FUNCTION_BLOCK ProductionRateFbt (* Composite Function Block Type *)
  (* Standard: 61499-2 *)
  (* Version 0.0, 2018-10-14, 4DIAC-IDE, 4DIAC-Consortium *)
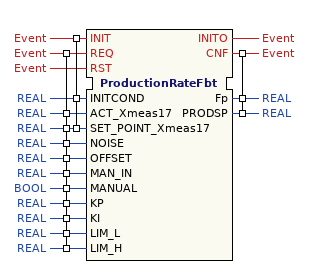
  EVENT_INPUT
    INIT WITH INITCOND, SET_POINT_Xmeas17; (* Initialization Request *)
    REQ WITH ACT_Xmeas17, SET_POINT_Xmeas17, NOISE, OFFSET, MAN_IN, MANUAL, KP, KI, LIM_L, LIM_H; (* Normal Execution Request *)
    RST;
  END_EVENT
  EVENT_OUTPUT
    INITO; (* Initialization Confirm *)
    CNF WITH Fp, PRODSP; (* Execution Confirmation *)
  END_EVENT
  VAR_INPUT
    INITCOND : REAL;
    ACT_Xmeas17 : REAL;
    SET_POINT_Xmeas17 : REAL;
    NOISE : REAL;
    OFFSET : REAL;
    MAN_IN : REAL;
    MANUAL : BOOL;
    KP : REAL;
    KI : REAL;
    LIM_L : REAL;
    LIM_H : REAL;
  END_VAR
  VAR_OUTPUT
    Fp : REAL;
    PRODSP : REAL;
  END_VAR
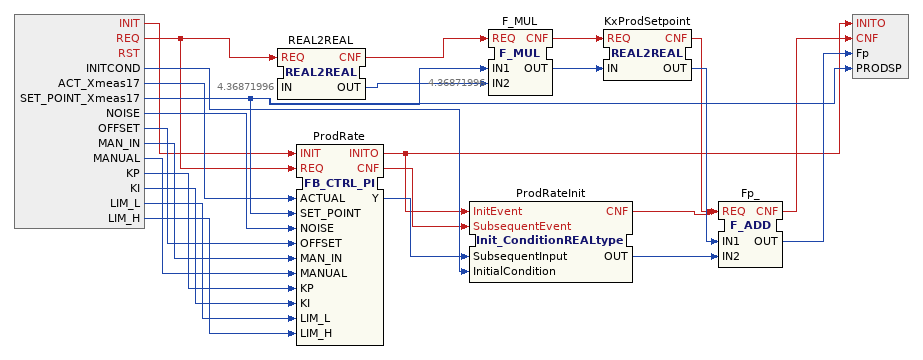
  FBS
    ProdRate : FB_CTRL_PI;
    F_MUL : F_MUL(IN2 := 4.36871996);
    KxProdSetpoint : REAL2REAL;
    ProdRateInit : Init_ConditionREALtype;
    Fp_ : F_ADD;
    REAL2REAL : REAL2REAL(IN := 4.36871996);
  END_FBS
  EVENT_CONNECTIONS
    INIT TO ProdRate.INIT;
    ProdRate.INITO TO ProdRateInit.InitEvent;
    ProdRate.CNF TO ProdRateInit.SubsequentEvent;
    REQ TO ProdRate.REQ;
    F_MUL.CNF TO KxProdSetpoint.REQ;
    KxProdSetpoint.CNF TO Fp_.REQ;
    ProdRateInit.CNF TO Fp_.REQ;
    Fp_.CNF TO CNF;
    ProdRate.INITO TO INITO;
    REAL2REAL.CNF TO F_MUL.REQ;
    REQ TO REAL2REAL.REQ;
  END_CONNECTIONS
  DATA_CONNECTIONS
    ProdRate.Y TO ProdRateInit.SubsequentInput;
    ACT_Xmeas17 TO ProdRate.ACTUAL;
    SET_POINT_Xmeas17 TO ProdRate.SET_POINT;
    SET_POINT_Xmeas17 TO F_MUL.IN1;
    F_MUL.OUT TO KxProdSetpoint.IN;
    KxProdSetpoint.OUT TO Fp_.IN1;
    ProdRateInit.OUT TO Fp_.IN2;
    Fp_.OUT TO Fp;
    NOISE TO ProdRate.NOISE;
    OFFSET TO ProdRate.OFFSET;
    MAN_IN TO ProdRate.MAN_IN;
    MANUAL TO ProdRate.MANUAL;
    KP TO ProdRate.KP;
    KI TO ProdRate.KI;
    LIM_L TO ProdRate.LIM_L;
    LIM_H TO ProdRate.LIM_H;
    SET_POINT_Xmeas17 TO PRODSP;
    INITCOND TO ProdRateInit.InitialCondition;
    REAL2REAL.OUT TO F_MUL.IN2;
  END_CONNECTIONS
END_FUNCTION_BLOCK
